{attribute 'GeneratedUsingTerminal: EL3681-0000-0018'}
{attribute addProperty BoxType "EL3681-0000-0018"}
{attribute addProperty Id "SettingsAT %I*Settings_24C049402"}
{attribute addProperty CRC "3183439273"}
{attribute addProperty Size "2"}
TYPE SAI_Range_BDBF6DA9 :
STRUCT
	{attribute addProperty Name "Settings"}
	Settings AT %I* : Settings_24C04940;
END_STRUCT
END_TYPE

(* stored: Version 1.2.0.0, ProductVersion 3.1.4024.9
   DUT SAI_Range_BDBF6DA9: Id {e4365ba7-4f45-4fc5-b3e5-3a26aa5893ff} *)
